{attribute 'GeneratedUsingTerminal: EL2535-0000-0016'}
{attribute addProperty BoxType "EL2535-0000-0016"}
{attribute addProperty Id "ControlAT %Q*Control_254441A53PWM_outputAT %Q*INT2"}
{attribute addProperty CRC "1676763876"}
{attribute addProperty Size "5"}
TYPE PWM_Control_Channel_63F162E4 EXTENDS OutputBase_10CEE7DE :
STRUCT
	{attribute addProperty Name "Control"}
	Control AT %Q* : Control_254441A5;
	{attribute addProperty Name "PWM_output"}
	PWM_output AT %Q* : INT;
END_STRUCT
END_TYPE

(* stored: Version 1.2.0.0, ProductVersion 3.1.4024.11
   DUT PWM_Control_Channel_63F162E4: Id {eeeae138-0ed4-4766-b13c-de98c3c96432} *)
